FUNCTION_BLOCK XARM5_ROBOT
  {SET_ATTRIBUTE(OpcUa, POINT.STARTPOINT)}
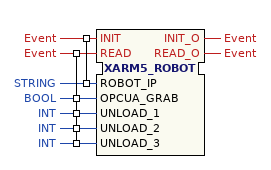
  EVENT_INPUT
    INIT WITH ROBOT_IP;
    READ WITH OPCUA_GRAB, UNLOAD_1, UNLOAD_2, UNLOAD_3;
  END_EVENT
  EVENT_OUTPUT
    INIT_O;
    READ_O;
  END_EVENT
  VAR_INPUT
    ROBOT_IP : STRING; {SET_ATTRIBUTE(OpcUa, Variable.RUN)}
    OPCUA_GRAB : BOOL; {SET_ATTRIBUTE(OpcUa, Variable.RUN)}
    UNLOAD_1 : INT; {SET_ATTRIBUTE(OpcUa, Variable.RUN)}
    UNLOAD_2 : INT; {SET_ATTRIBUTE(OpcUa, Variable.RUN)}
    UNLOAD_3 : INT; {SET_ATTRIBUTE(OpcUa, Variable.RUN)}
  END_VAR
END_FUNCTION_BLOCK
